(* Logix 5000 project; controller Turck_IOLink_All_Full_AOIs_V0_1 vendor 1 type 14 code 176 rev 32.11; software revision 32.00; part 5 of 7 *)
(* tags used below, declared in another part *)
   Error_DINT : DINT;
   Write : DINT;
(* Turck_PS510_10V_Full, continued *)

ROUTINE Prescan   (* ladder *)
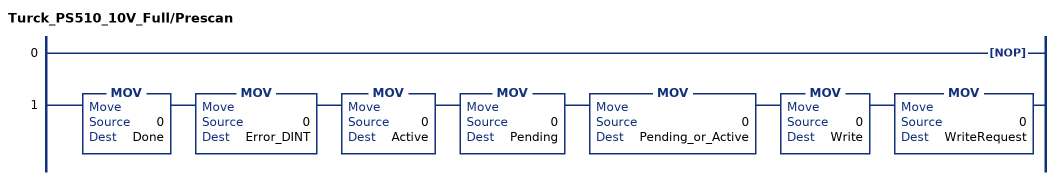
   0: NOP();
   1: MOV(0,Done)MOV(0,Error_DINT)MOV(0,Active)MOV(0,Pending)MOV(0,Pending_or_Active)MOV(0,Write)MOV(0,WriteRequest);
END_ROUTINE
END_ADD_ON_INSTRUCTION

ADD_ON_INSTRUCTION Turck_TBIL_M1_16DXP_Full   (* revision 1.0 *)
VAR_INPUT
   Port : INT; {required}
END_VAR
VAR_IN_OUT
   Common_Data : Turck_IOLink_Common_Data; {required}
END_VAR
VAR_OUTPUT
   Input_1A : BOOL; {visible}
   Input_1B : BOOL; {visible}
   Input_2A : BOOL; {visible}
   Input_2B : BOOL; {visible}
   Input_3A : BOOL; {visible}
   Input_3B : BOOL; {visible}
   Input_4A : BOOL; {visible}
   Input_4B : BOOL; {visible}
   Input_5A : BOOL; {visible}
   Input_5B : BOOL; {visible}
   Input_6A : BOOL; {visible}
   Input_6B : BOOL; {visible}
   Input_7A : BOOL; {visible}
   Input_7B : BOOL; {visible}
   Input_8A : BOOL; {visible}
   Input_8B : BOOL; {visible}
END_VAR
VAR_INPUT
   Output_1A : BOOL; {visible}
   Output_1B : BOOL; {visible}
   Output_2A : BOOL; {visible}
   Output_2B : BOOL; {visible}
   Output_3A : BOOL; {visible}
   Output_3B : BOOL; {visible}
   Output_4A : BOOL; {visible}
   Output_4B : BOOL; {visible}
   Output_5A : BOOL; {visible}
   Output_5B : BOOL; {visible}
   Output_6A : BOOL; {visible}
   Output_6B : BOOL; {visible}
   Output_7A : BOOL; {visible}
   Output_7B : BOOL; {visible}
   Output_8A : BOOL; {visible}
   Output_8B : BOOL; {visible}
END_VAR
VAR_OUTPUT
   Wrong_or_Missing_Device : BOOL; {visible}
END_VAR
VAR
   Port_Less_One : INT; {access None}
   One : SINT; {access None}
   Port_Bit : SINT; {access None}
   Two : DINT; {access None}
END_VAR

ROUTINE Logic   (* ladder *)
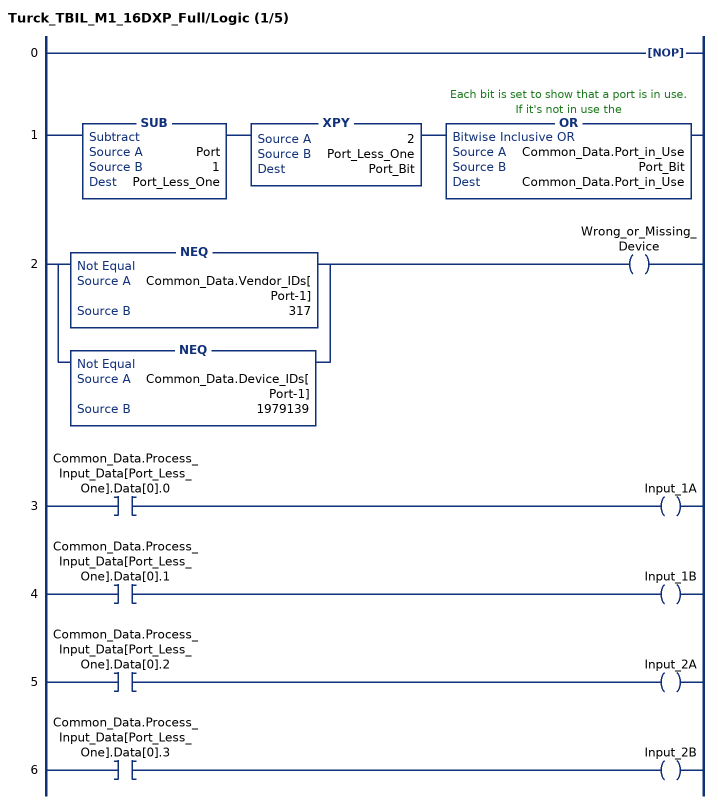
   0: NOP();
   1: SUB(Port,1,Port_Less_One)XPY(2,Port_Less_One,Port_Bit)OR(Common_Data.Port_in_Use,Port_Bit,Common_Data.Port_in_Use);
   2: [NEQ(Common_Data.Vendor_IDs[Port-1],317) ,NEQ(Common_Data.Device_IDs[Port-1],1979139) ]OTE(Wrong_or_Missing_Device);
   3: XIC(Common_Data.Process_Input_Data[Port_Less_One].Data[0].0)OTE(Input_1A);
   4: XIC(Common_Data.Process_Input_Data[Port_Less_One].Data[0].1)OTE(Input_1B);
   5: XIC(Common_Data.Process_Input_Data[Port_Less_One].Data[0].2)OTE(Input_2A);
   6: XIC(Common_Data.Process_Input_Data[Port_Less_One].Data[0].3)OTE(Input_2B);
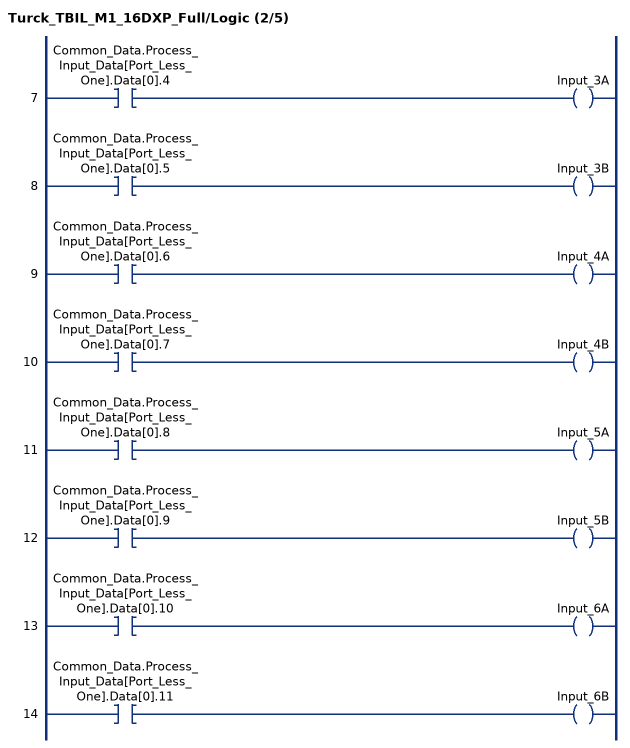
   7: XIC(Common_Data.Process_Input_Data[Port_Less_One].Data[0].4)OTE(Input_3A);
   8: XIC(Common_Data.Process_Input_Data[Port_Less_One].Data[0].5)OTE(Input_3B);
   9: XIC(Common_Data.Process_Input_Data[Port_Less_One].Data[0].6)OTE(Input_4A);
   10: XIC(Common_Data.Process_Input_Data[Port_Less_One].Data[0].7)OTE(Input_4B);
   11: XIC(Common_Data.Process_Input_Data[Port_Less_One].Data[0].8)OTE(Input_5A);
   12: XIC(Common_Data.Process_Input_Data[Port_Less_One].Data[0].9)OTE(Input_5B);
   13: XIC(Common_Data.Process_Input_Data[Port_Less_One].Data[0].10)OTE(Input_6A);
   14: XIC(Common_Data.Process_Input_Data[Port_Less_One].Data[0].11)OTE(Input_6B);
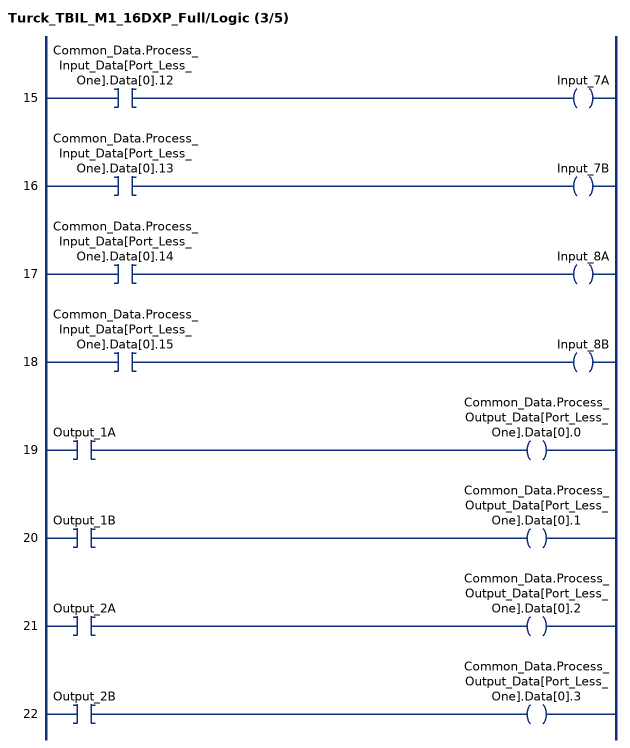
   15: XIC(Common_Data.Process_Input_Data[Port_Less_One].Data[0].12)OTE(Input_7A);
   16: XIC(Common_Data.Process_Input_Data[Port_Less_One].Data[0].13)OTE(Input_7B);
   17: XIC(Common_Data.Process_Input_Data[Port_Less_One].Data[0].14)OTE(Input_8A);
   18: XIC(Common_Data.Process_Input_Data[Port_Less_One].Data[0].15)OTE(Input_8B);
   19: XIC(Output_1A)OTE(Common_Data.Process_Output_Data[Port_Less_One].Data[0].0);
   20: XIC(Output_1B)OTE(Common_Data.Process_Output_Data[Port_Less_One].Data[0].1);
   21: XIC(Output_2A)OTE(Common_Data.Process_Output_Data[Port_Less_One].Data[0].2);
   22: XIC(Output_2B)OTE(Common_Data.Process_Output_Data[Port_Less_One].Data[0].3);
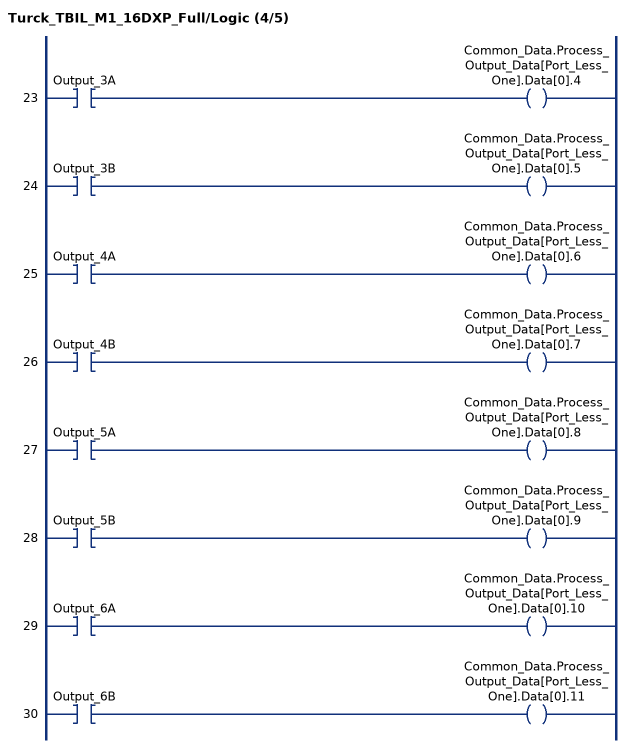
   23: XIC(Output_3A)OTE(Common_Data.Process_Output_Data[Port_Less_One].Data[0].4);
   24: XIC(Output_3B)OTE(Common_Data.Process_Output_Data[Port_Less_One].Data[0].5);
   25: XIC(Output_4A)OTE(Common_Data.Process_Output_Data[Port_Less_One].Data[0].6);
   26: XIC(Output_4B)OTE(Common_Data.Process_Output_Data[Port_Less_One].Data[0].7);
   27: XIC(Output_5A)OTE(Common_Data.Process_Output_Data[Port_Less_One].Data[0].8);
   28: XIC(Output_5B)OTE(Common_Data.Process_Output_Data[Port_Less_One].Data[0].9);
   29: XIC(Output_6A)OTE(Common_Data.Process_Output_Data[Port_Less_One].Data[0].10);
   30: XIC(Output_6B)OTE(Common_Data.Process_Output_Data[Port_Less_One].Data[0].11);
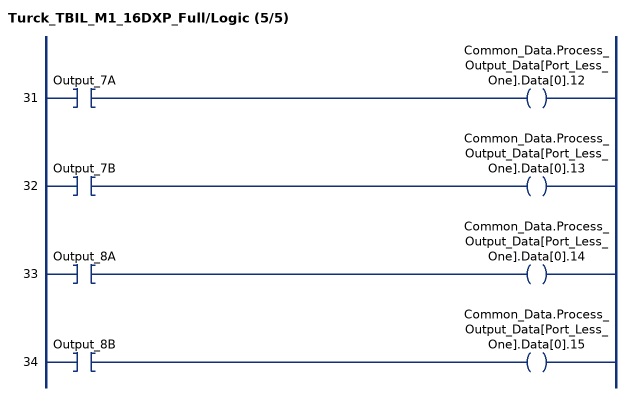
   31: XIC(Output_7A)OTE(Common_Data.Process_Output_Data[Port_Less_One].Data[0].12);
   32: XIC(Output_7B)OTE(Common_Data.Process_Output_Data[Port_Less_One].Data[0].13);
   33: XIC(Output_8A)OTE(Common_Data.Process_Output_Data[Port_Less_One].Data[0].14);
   34: XIC(Output_8B)OTE(Common_Data.Process_Output_Data[Port_Less_One].Data[0].15);
END_ROUTINE
END_ADD_ON_INSTRUCTION

ADD_ON_INSTRUCTION Universal_Device_Info   (* revision 1.0, ExecutePrescan *)
VAR_INPUT
   Port : INT; {required}
END_VAR
VAR_IN_OUT
   Common_Data : Turck_IOLink_Common_Data; {required}
END_VAR
VAR_INPUT
   Write_Application_Specific_Tag : BOOL;
END_VAR
VAR_IN_OUT
   Universal_IOLink_Info : Universal_IOLink_Info; {required}
END_VAR
VAR
   StartupDone : BOOL; {access None}
   Done : DINT; {access None}
   Error : DINT; {access None}
   Active : DINT; {access None}
   Pending : DINT; {access None}
   Pending_or_Active : DINT; {access None}
   StartupCount : DINT; {access None}
   MyTicketNum : DINT[32]; {access None}
   Read_ONS : DINT; {access None}
   ReadRequest : DINT; {access None}
   Read : DINT; {access None}
   DoneCount : DINT; {access None}
   Status : DINT; {access None}
   ErrorCount : DINT; {access None}
   Prev_Vendor_ID : INT; {access None}
   Update_Data : BOOL; {access None}
   Reset : BOOL; {access None}
   Write_ONS : DINT; {access None}
   WriteRequest : DINT; {access None}
END_VAR

ROUTINE Logic   (* ladder *)
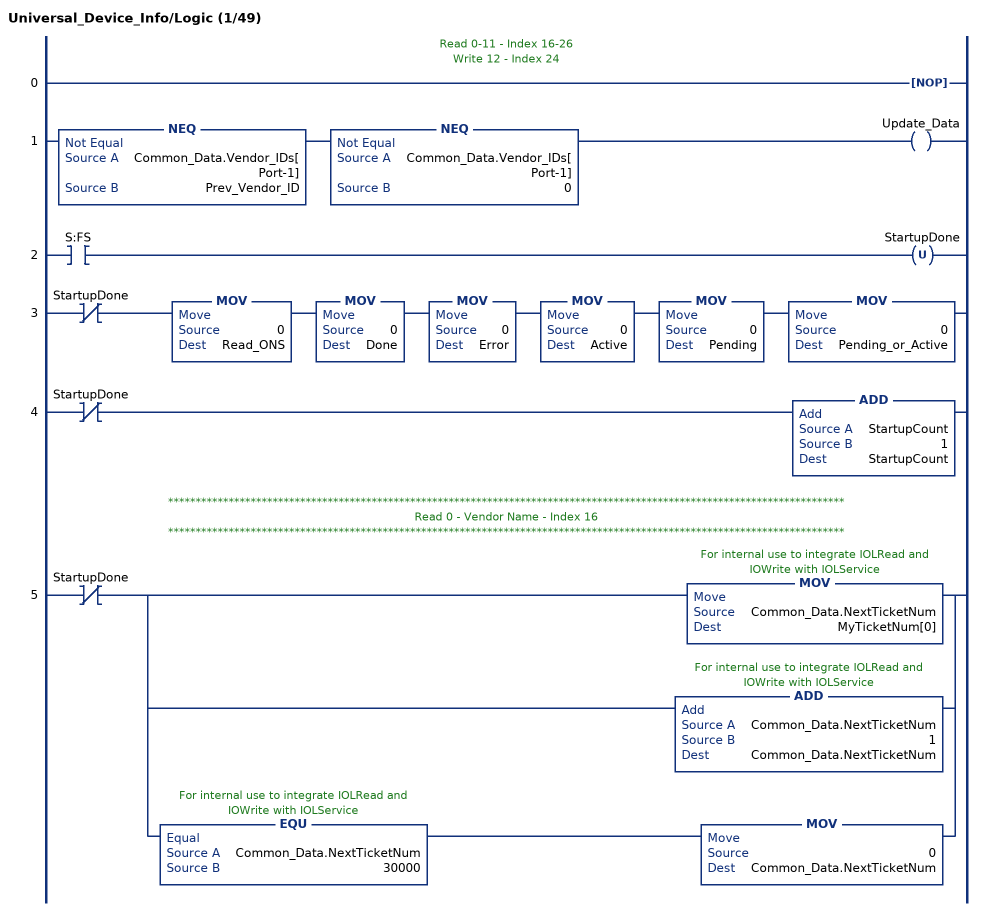
   // Read 0-11 - Index 16-26
   // Write 12 - Index 24
   0: NOP();
   1: NEQ(Common_Data.Vendor_IDs[Port-1],Prev_Vendor_ID)NEQ(Common_Data.Vendor_IDs[Port-1],0)OTE(Update_Data);
   2: XIC(S:FS)OTU(StartupDone);
   3: XIO(StartupDone)MOV(0,Read_ONS)MOV(0,Done)MOV(0,Error)MOV(0,Active)MOV(0,Pending)MOV(0,Pending_or_Active);
   4: XIO(StartupDone)ADD(StartupCount,1,StartupCount);
   // ***************************************************************************************************************************
   // Read 0 - Vendor Name - Index 16
   // ***************************************************************************************************************************
   5: XIO(StartupDone)[MOV(Common_Data.NextTicketNum,MyTicketNum[0]) ,ADD(Common_Data.NextTicketNum,1,Common_Data.NextTicketNum) ,EQU(Common_Data.NextTicketNum,30000) MOV(0,Common_Data.NextTicketNum) ];
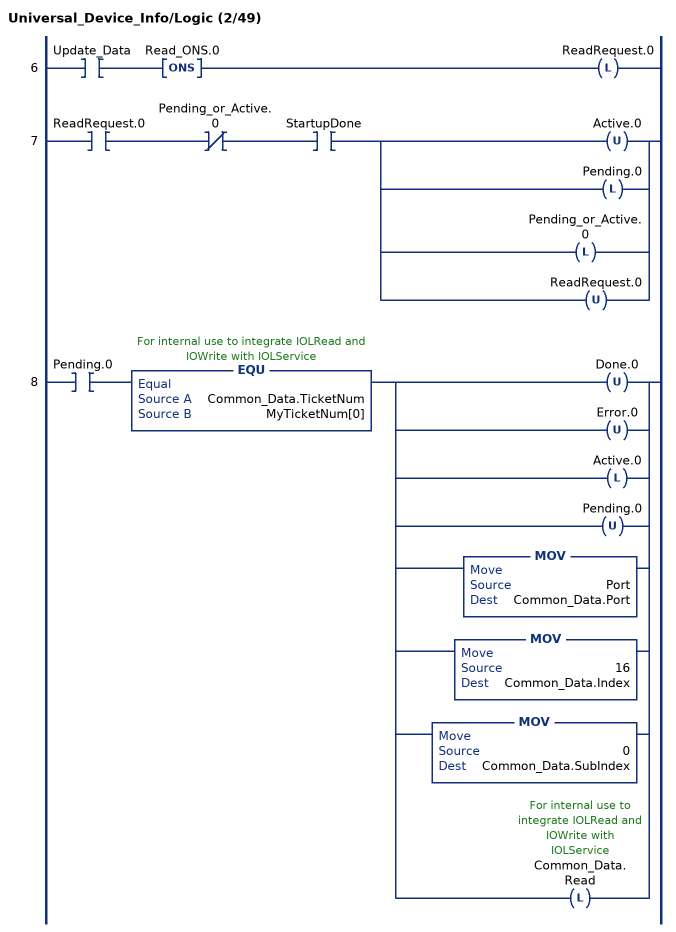
   6: XIC(Update_Data)ONS(Read_ONS.0)OTL(ReadRequest.0);
   7: XIC(ReadRequest.0)XIO(Pending_or_Active.0)XIC(StartupDone)[OTU(Active.0) ,OTL(Pending.0) ,OTL(Pending_or_Active.0) ,OTU(ReadRequest.0) ];
   8: XIC(Pending.0)EQU(Common_Data.TicketNum,MyTicketNum[0])[OTU(Done.0) ,OTU(Error.0) ,OTL(Active.0) ,OTU(Pending.0) ,MOV(Port,Common_Data.Port) ,MOV(16,Common_Data.Index) ,MOV(0,Common_Data.SubIndex) ,OTL(Common_Data.Read) ];
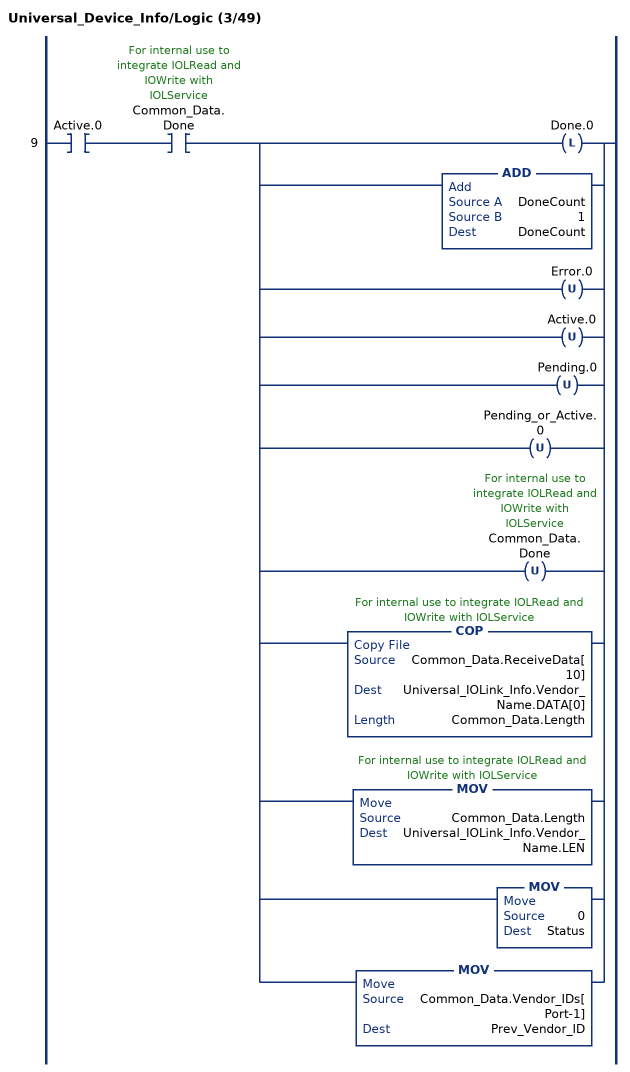
   9: XIC(Active.0)XIC(Common_Data.Done)[OTL(Done.0) ,ADD(DoneCount,1,DoneCount) ,OTU(Error.0) ,OTU(Active.0) ,OTU(Pending.0) ,OTU(Pending_or_Active.0) ,OTU(Common_Data.Done) ,COP(Common_Data.ReceiveData[10],Universal_IOLink_Info.Vendor_Name.DATA[0],Common_Data.Length) ,MOV(Common_Data.Length,Universal_IOLink_Info.Vendor_Name.LEN) ,MOV(0,Status) ,MOV(Common_Data.Vendor_IDs[Port-1],Prev_Vendor_ID) ];
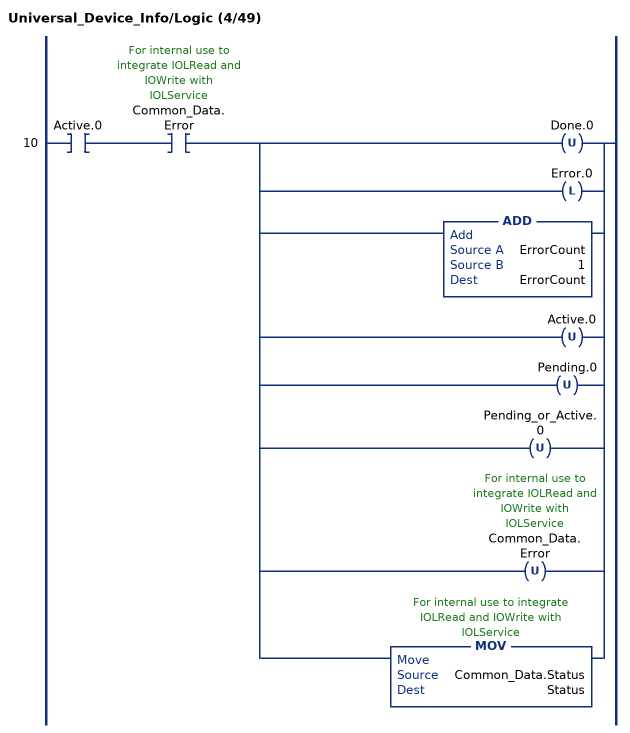
   10: XIC(Active.0)XIC(Common_Data.Error)[OTU(Done.0) ,OTL(Error.0) ,ADD(ErrorCount,1,ErrorCount) ,OTU(Active.0) ,OTU(Pending.0) ,OTU(Pending_or_Active.0) ,OTU(Common_Data.Error) ,MOV(Common_Data.Status,Status) ];
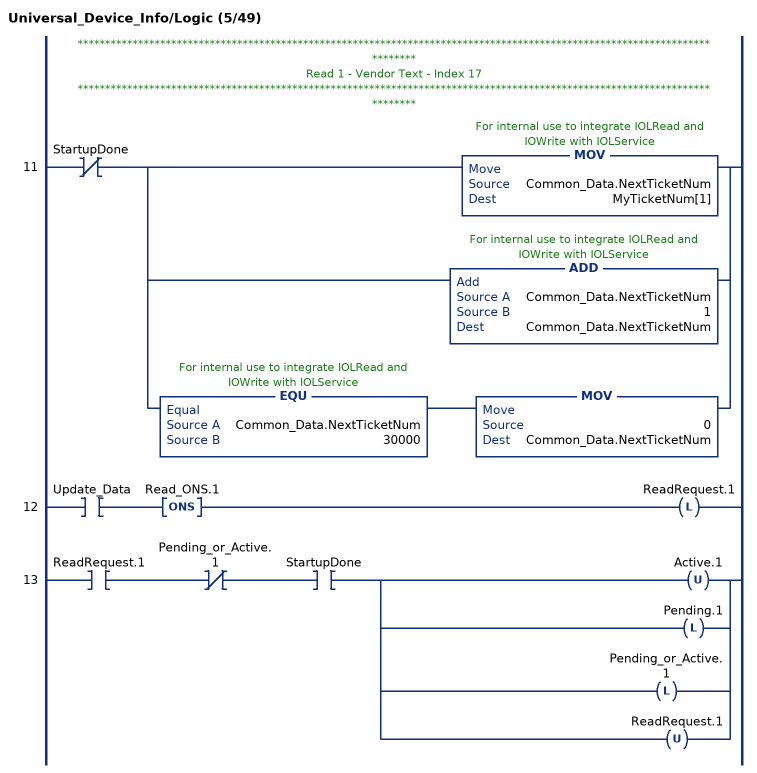
   // ***************************************************************************************************************************
   // Read 1 - Vendor Text - Index 17
   // ***************************************************************************************************************************
   11: XIO(StartupDone)[MOV(Common_Data.NextTicketNum,MyTicketNum[1]) ,ADD(Common_Data.NextTicketNum,1,Common_Data.NextTicketNum) ,EQU(Common_Data.NextTicketNum,30000) MOV(0,Common_Data.NextTicketNum) ];
   12: XIC(Update_Data)ONS(Read_ONS.1)OTL(ReadRequest.1);
   13: XIC(ReadRequest.1)XIO(Pending_or_Active.1)XIC(StartupDone)[OTU(Active.1) ,OTL(Pending.1) ,OTL(Pending_or_Active.1) ,OTU(ReadRequest.1) ];
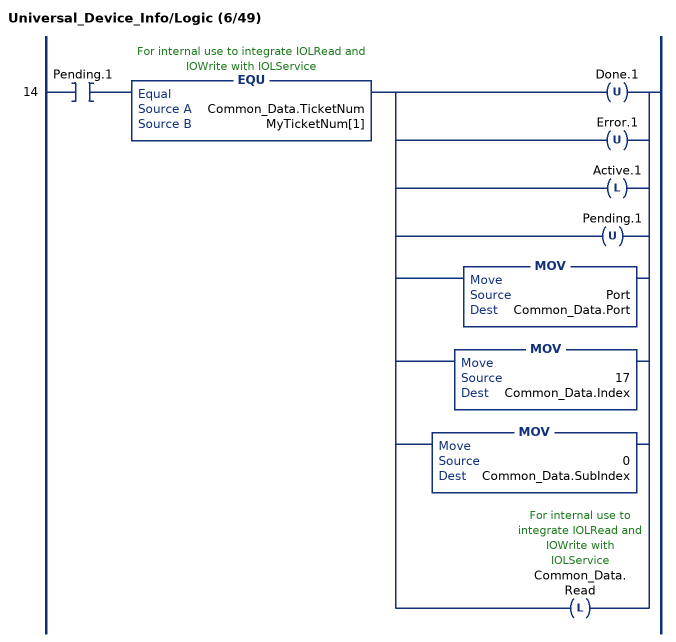
   14: XIC(Pending.1)EQU(Common_Data.TicketNum,MyTicketNum[1])[OTU(Done.1) ,OTU(Error.1) ,OTL(Active.1) ,OTU(Pending.1) ,MOV(Port,Common_Data.Port) ,MOV(17,Common_Data.Index) ,MOV(0,Common_Data.SubIndex) ,OTL(Common_Data.Read) ];
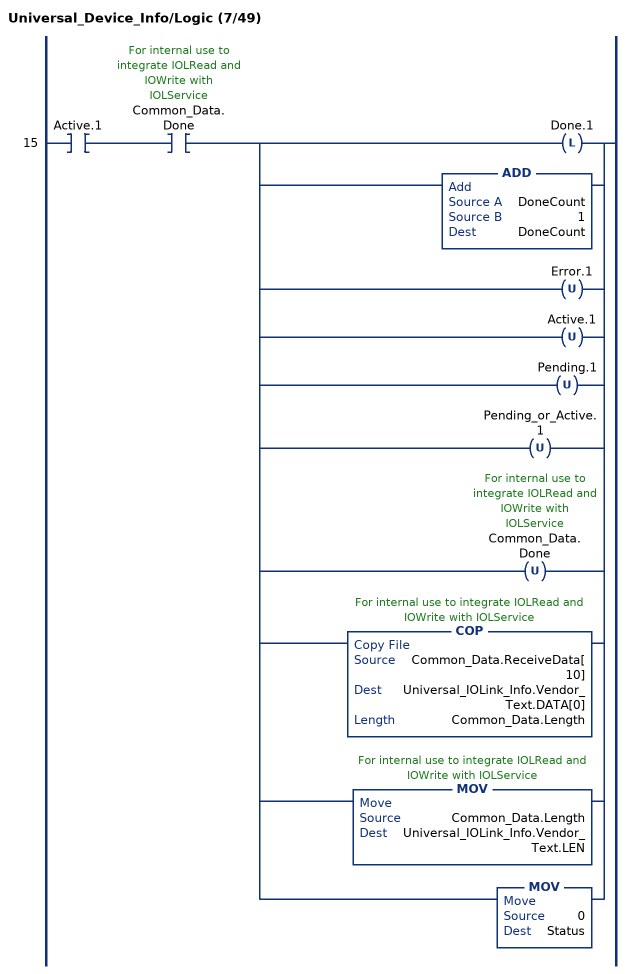
   15: XIC(Active.1)XIC(Common_Data.Done)[OTL(Done.1) ,ADD(DoneCount,1,DoneCount) ,OTU(Error.1) ,OTU(Active.1) ,OTU(Pending.1) ,OTU(Pending_or_Active.1) ,OTU(Common_Data.Done) ,COP(Common_Data.ReceiveData[10],Universal_IOLink_Info.Vendor_Text.DATA[0],Common_Data.Length) ,MOV(Common_Data.Length,Universal_IOLink_Info.Vendor_Text.LEN) ,MOV(0,Status) ];
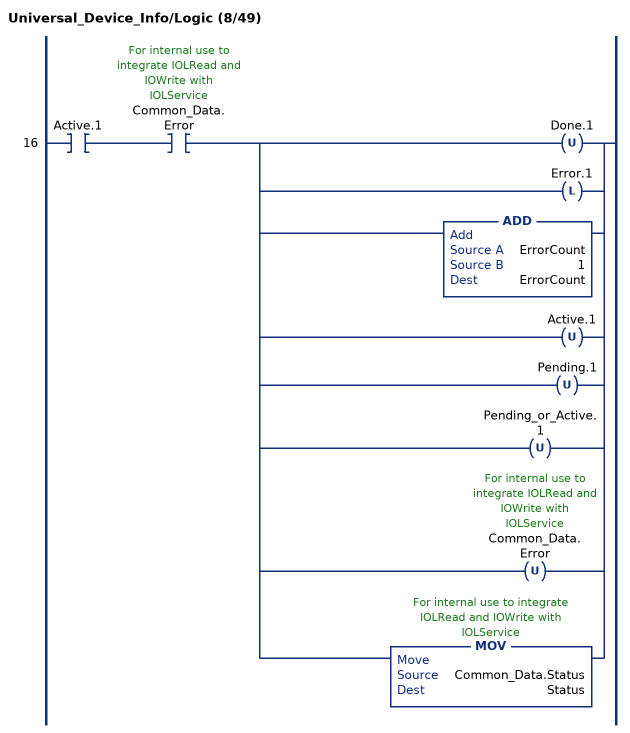
   16: XIC(Active.1)XIC(Common_Data.Error)[OTU(Done.1) ,OTL(Error.1) ,ADD(ErrorCount,1,ErrorCount) ,OTU(Active.1) ,OTU(Pending.1) ,OTU(Pending_or_Active.1) ,OTU(Common_Data.Error) ,MOV(Common_Data.Status,Status) ];
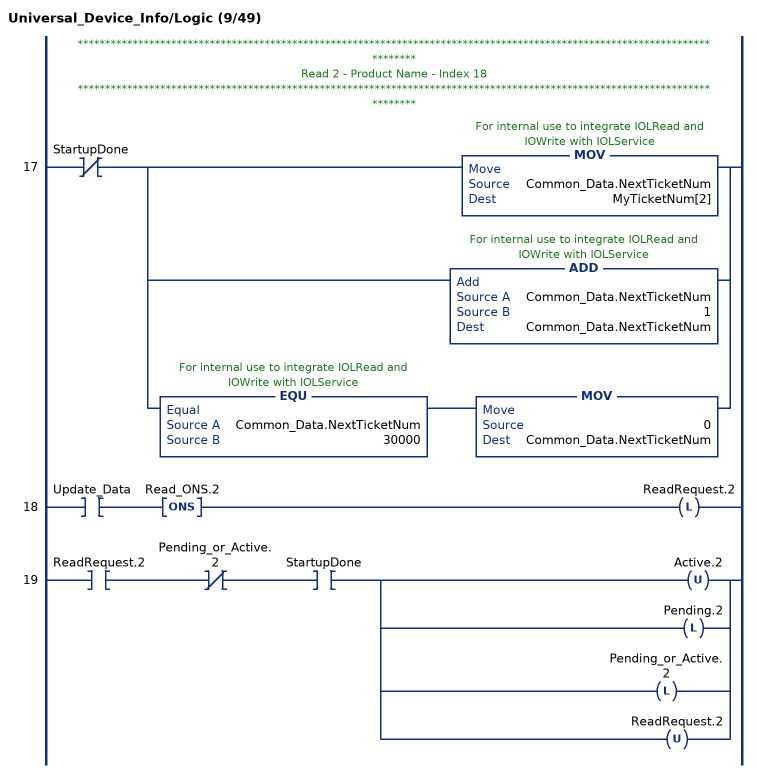
   // ***************************************************************************************************************************
   // Read 2 - Product Name - Index 18
   // ***************************************************************************************************************************
   17: XIO(StartupDone)[MOV(Common_Data.NextTicketNum,MyTicketNum[2]) ,ADD(Common_Data.NextTicketNum,1,Common_Data.NextTicketNum) ,EQU(Common_Data.NextTicketNum,30000) MOV(0,Common_Data.NextTicketNum) ];
   18: XIC(Update_Data)ONS(Read_ONS.2)OTL(ReadRequest.2);
   19: XIC(ReadRequest.2)XIO(Pending_or_Active.2)XIC(StartupDone)[OTU(Active.2) ,OTL(Pending.2) ,OTL(Pending_or_Active.2) ,OTU(ReadRequest.2) ];
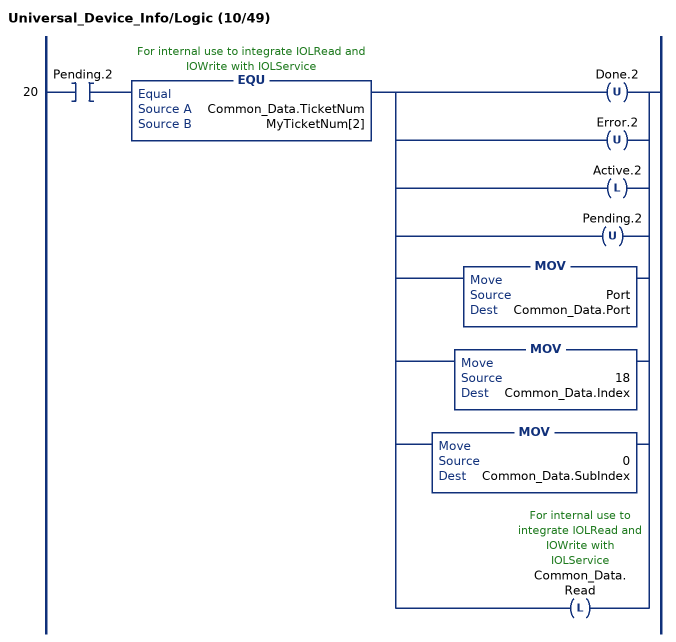
   20: XIC(Pending.2)EQU(Common_Data.TicketNum,MyTicketNum[2])[OTU(Done.2) ,OTU(Error.2) ,OTL(Active.2) ,OTU(Pending.2) ,MOV(Port,Common_Data.Port) ,MOV(18,Common_Data.Index) ,MOV(0,Common_Data.SubIndex) ,OTL(Common_Data.Read) ];
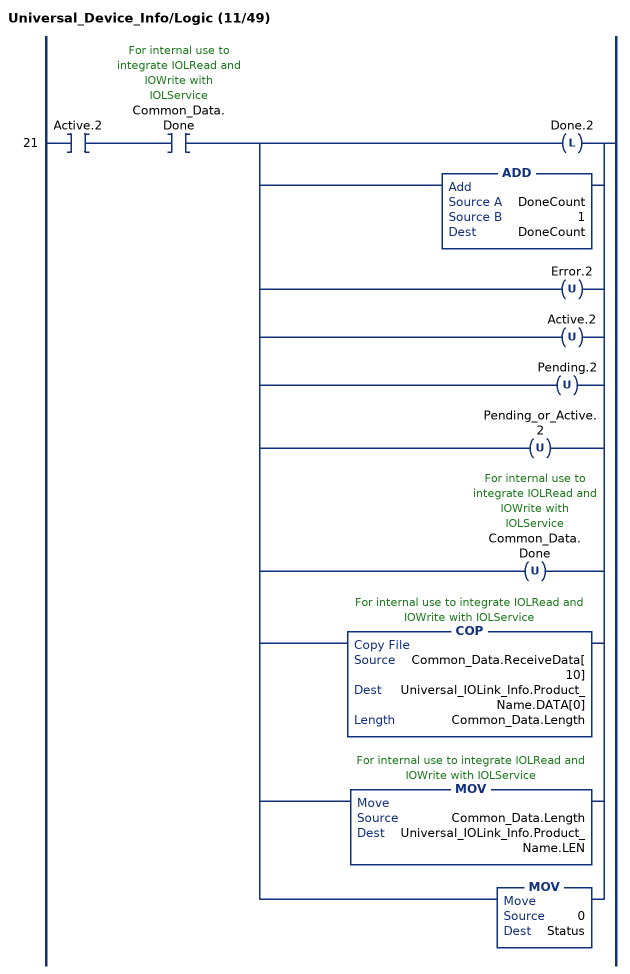
   21: XIC(Active.2)XIC(Common_Data.Done)[OTL(Done.2) ,ADD(DoneCount,1,DoneCount) ,OTU(Error.2) ,OTU(Active.2) ,OTU(Pending.2) ,OTU(Pending_or_Active.2) ,OTU(Common_Data.Done) ,COP(Common_Data.ReceiveData[10],Universal_IOLink_Info.Product_Name.DATA[0],Common_Data.Length) ,MOV(Common_Data.Length,Universal_IOLink_Info.Product_Name.LEN) ,MOV(0,Status) ];
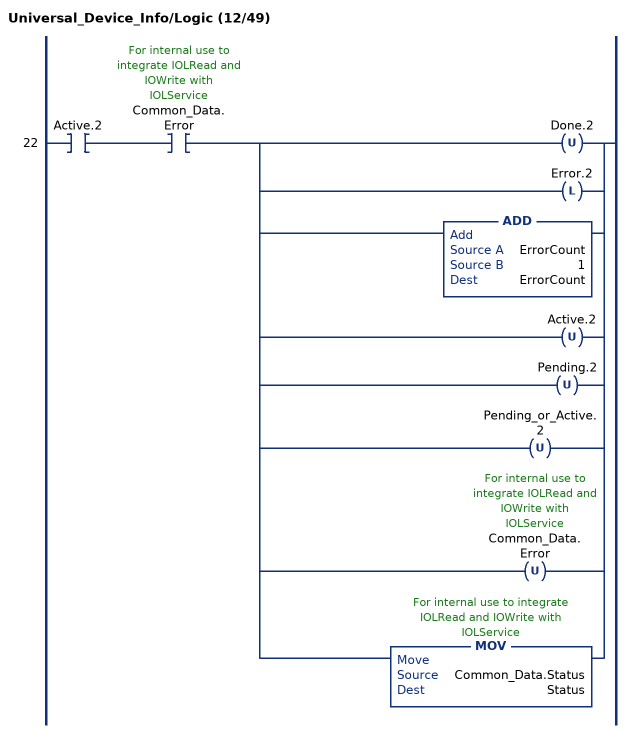
   22: XIC(Active.2)XIC(Common_Data.Error)[OTU(Done.2) ,OTL(Error.2) ,ADD(ErrorCount,1,ErrorCount) ,OTU(Active.2) ,OTU(Pending.2) ,OTU(Pending_or_Active.2) ,OTU(Common_Data.Error) ,MOV(Common_Data.Status,Status) ];
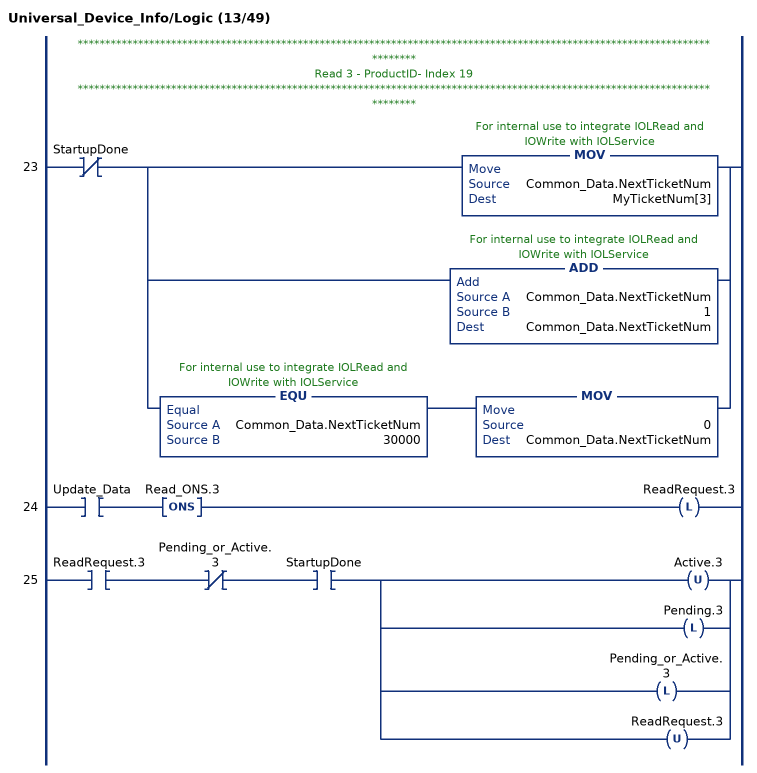
   // ***************************************************************************************************************************
   // Read 3 - ProductID- Index 19
   // ***************************************************************************************************************************
   23: XIO(StartupDone)[MOV(Common_Data.NextTicketNum,MyTicketNum[3]) ,ADD(Common_Data.NextTicketNum,1,Common_Data.NextTicketNum) ,EQU(Common_Data.NextTicketNum,30000) MOV(0,Common_Data.NextTicketNum) ];
   24: XIC(Update_Data)ONS(Read_ONS.3)OTL(ReadRequest.3);
   25: XIC(ReadRequest.3)XIO(Pending_or_Active.3)XIC(StartupDone)[OTU(Active.3) ,OTL(Pending.3) ,OTL(Pending_or_Active.3) ,OTU(ReadRequest.3) ];
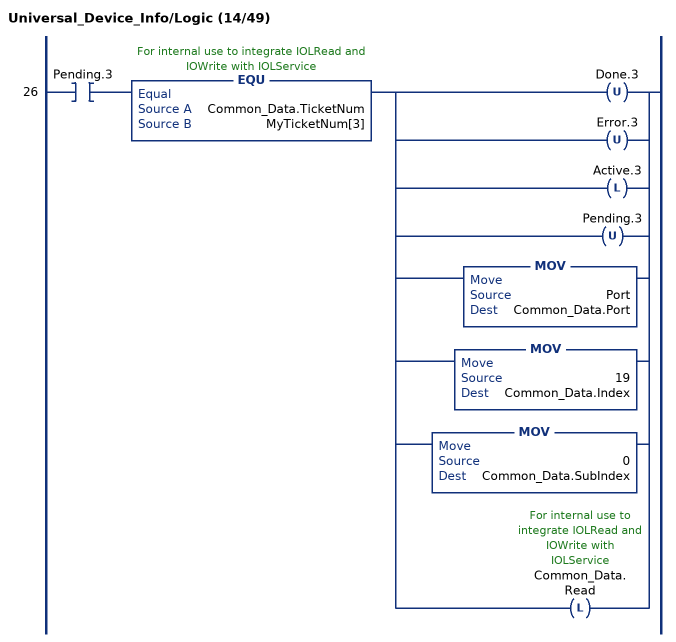
   26: XIC(Pending.3)EQU(Common_Data.TicketNum,MyTicketNum[3])[OTU(Done.3) ,OTU(Error.3) ,OTL(Active.3) ,OTU(Pending.3) ,MOV(Port,Common_Data.Port) ,MOV(19,Common_Data.Index) ,MOV(0,Common_Data.SubIndex) ,OTL(Common_Data.Read) ];
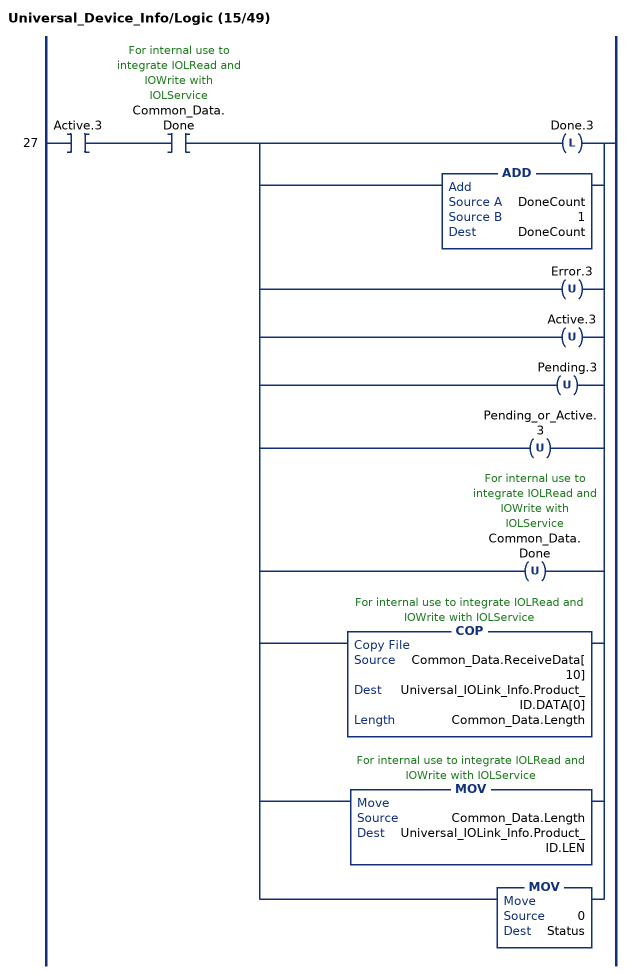
   27: XIC(Active.3)XIC(Common_Data.Done)[OTL(Done.3) ,ADD(DoneCount,1,DoneCount) ,OTU(Error.3) ,OTU(Active.3) ,OTU(Pending.3) ,OTU(Pending_or_Active.3) ,OTU(Common_Data.Done) ,COP(Common_Data.ReceiveData[10],Universal_IOLink_Info.Product_ID.DATA[0],Common_Data.Length) ,MOV(Common_Data.Length,Universal_IOLink_Info.Product_ID.LEN) ,MOV(0,Status) ];
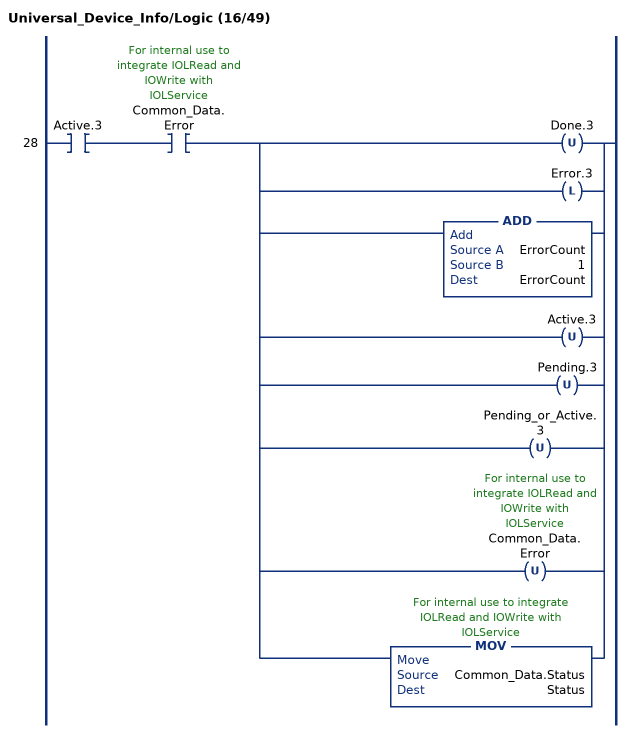
   28: XIC(Active.3)XIC(Common_Data.Error)[OTU(Done.3) ,OTL(Error.3) ,ADD(ErrorCount,1,ErrorCount) ,OTU(Active.3) ,OTU(Pending.3) ,OTU(Pending_or_Active.3) ,OTU(Common_Data.Error) ,MOV(Common_Data.Status,Status) ];
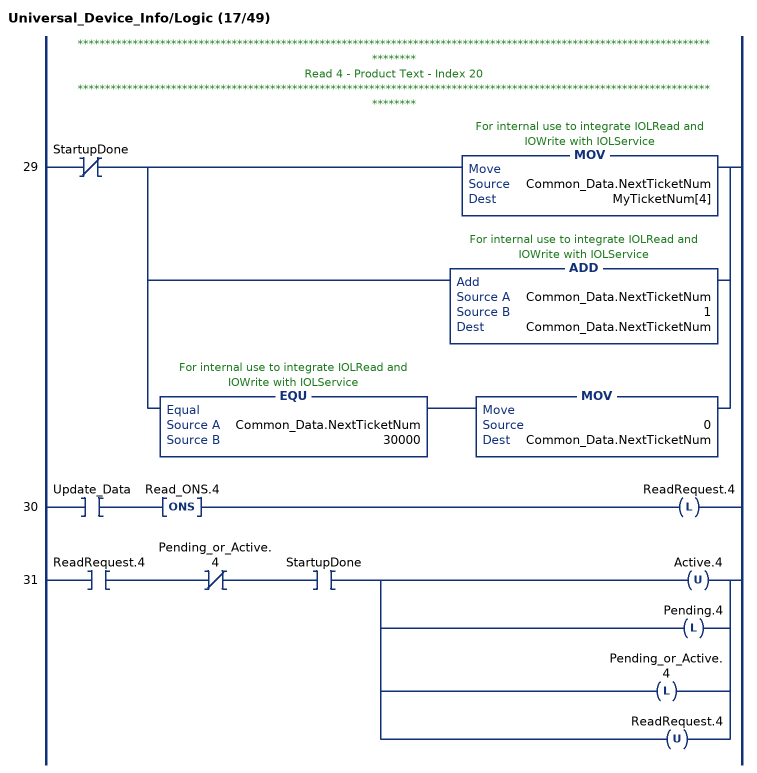
   // ***************************************************************************************************************************
   // Read 4 - Product Text - Index 20
   // ***************************************************************************************************************************
   29: XIO(StartupDone)[MOV(Common_Data.NextTicketNum,MyTicketNum[4]) ,ADD(Common_Data.NextTicketNum,1,Common_Data.NextTicketNum) ,EQU(Common_Data.NextTicketNum,30000) MOV(0,Common_Data.NextTicketNum) ];
   30: XIC(Update_Data)ONS(Read_ONS.4)OTL(ReadRequest.4);
   31: XIC(ReadRequest.4)XIO(Pending_or_Active.4)XIC(StartupDone)[OTU(Active.4) ,OTL(Pending.4) ,OTL(Pending_or_Active.4) ,OTU(ReadRequest.4) ];
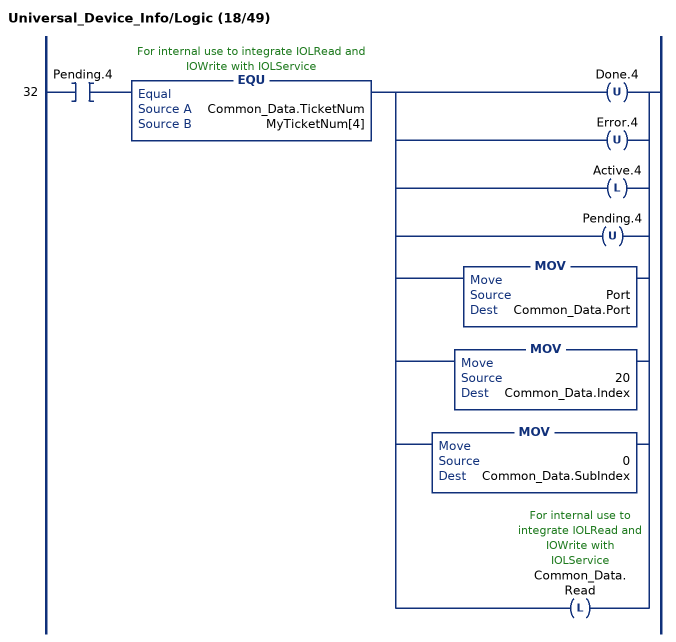
   32: XIC(Pending.4)EQU(Common_Data.TicketNum,MyTicketNum[4])[OTU(Done.4) ,OTU(Error.4) ,OTL(Active.4) ,OTU(Pending.4) ,MOV(Port,Common_Data.Port) ,MOV(20,Common_Data.Index) ,MOV(0,Common_Data.SubIndex) ,OTL(Common_Data.Read) ];
